{attribute addProperty BoxType "AX8206-0000-0041-0041"}
{attribute addProperty Id "AdsAddrAT %I*AMSADDR6480DcOutputShiftAT %I*DINT3240DcInputShiftAT %I*DINT3240AoeNetIdAT %I*AMSNETID4860Chn0AT %I*USINT810Chn1AT %I*USINT810StateAT %I*UINT1620"}
{attribute addProperty CRC "388463706"}
{attribute addProperty SizeInBites "208"}
{attribute addProperty SizeInBytes "26"}
TYPE InfoData_17277C5A :
STRUCT
	{attribute addProperty Name "AdsAddr"}
	AdsAddr AT %I* : AMSADDR;
	{attribute addProperty Name "DcOutputShift"}
	DcOutputShift AT %I* : DINT;
	{attribute addProperty Name "DcInputShift"}
	DcInputShift AT %I* : DINT;
	{attribute addProperty Name "AoeNetId"}
	AoeNetId AT %I* : AMSNETID;
	{attribute addProperty Name "Chn0"}
	Chn0 AT %I* : USINT;
	{attribute addProperty Name "Chn1"}
	Chn1 AT %I* : USINT;
	{attribute addProperty Name "State"}
	State AT %I* : UINT;
END_STRUCT
END_TYPE

(* stored: Version 1.2.0.0, ProductVersion 3.1.4024.9
   DUT InfoData_17277C5A: Id {7df2fe2c-1ee0-43cd-a01b-9aa901e2348c} *)
